Staubli VAL3: goHome.pjx

--- goHome.pjx ---
Parameters version=s7.8.3 stackSize=5000 millimeterUnit=true
Program file=_getP2PAngle.pgx
Program file=_getP2PDistance.pgx
Program file=_IsUseingBox.pgx
Program file=compteBox1Value.pgx
Program file=delete.pgx
Program file=editBigData.pgx
Program file=editSmlData.pgx
Program file=FCheckInBox1Pos.pgx
Program file=FCheckInBox2Pos.pgx
Program file=find.pgx
Program file=findInWhichBox1.pgx
Program file=FNearJt.pgx
Program file=getBoxSize.pgx
Program file=getEvent.pgx
Program file=getListTitle.pgx
Program file=getSizeItem.pgx
Program file=getTrajTool.pgx
Program file=GOHOME.pgx
Program file=goTo.pgx
Program file=HMI_setNewValue.pgx
Program file=HMI_setValue.pgx
Program file=initToSafePt.pgx
Program file=IsInTheSameBox.pgx
Program file=IsSetValue.pgx
Program file=IsUseSameTool.pgx
Program file=J_goTo.pgx
Program file=J_MoveTo.pgx
Program file=listAdd.pgx
Program file=loadMarkData.pgx
Program file=mark_All_Item.pgx
Program file=markItem.pgx
Program file=MoveTo.pgx
Program file=new.pgx
Program file=onSave.pgx
Program file=reveMarkItem.pgx
Data file=goHome.dtx
Library alias=sml path=./saveHomeBox/type1/type1.pjx
Library alias=big path=./saveHomeBox/type2/type2.pjx
Library alias=save path=./saveHomeBox/saveHomeBox.pjx
Library alias=language2 path=./language/language.pjx
Library alias=trajPt path=Disk://session/default/saveTraj/TRAJ/TRAJ.pjx
Library alias=saveData path=Disk://saveData/saveData.pjx
Library alias=jPt path=Disk://session/default/saveTraj/JPOINT/JPOINT.pjx
Library alias=use path=./userPage/userPage.pjx
Library alias=cycleStatus path=Disk://cycleStatus/cycleStatus.pjx
Library alias=tcp path=Disk://kernel/tool/tool.pjx
Library alias=language path=Disk://kernel/language/language.pjx
Library alias=jHome path=Disk://session/default/saveTraj/HOME/HOME.pjx
Type name=TrajSmallBox path=./template/TrajSmallBox/TrajSmallBox.pjx
Type name=TrajBigBox path=./template/TrajBigBox/TrajBigBox.pjx
Type name=TrajJoint path=Disk://kernel/template/TrajJoint/TrajJoint.pjx
Type name=Traies path=Disk://kernel/template/Traies/Traies.pjx

--- goHome.dtx ---
public TrajBigBox pRunBigPt
  [0]
    bool bJtEnabCheck[6]
    bool bMoveJHomeJoint
    bool bPosEnabCheck[3]
    jointRx jToHome
    num nIndexGun
    num nRobCtrlAreaNum[6]
    num nRobCtrlHJtsNum[12]
public TrajJoint tTrajJoint
  [0]
    num nIndexFrame
    num nIndexTool
    string sID = "qwer"
    TrajJointItem tData[2]
      [0]
        jointRx jJoint = {j1=-15.581719, j2=14.249611, j3=85.047741, j5=80.702759, j6=3.379944}
        TrajectoryItem tSuper
          [0]
            string comment
            num distance
            InstrItem iInstr[3]
              [0]
                string sData
                string sType
              [1]
                string sData
                string sType
              [2]
                string sData
                string sType
            num moveType
            num nMoveId
            num nStop
            num nTcpAction
            num nTime
            mdesc nom_speed = {tmax=9999, rmax=9999, leave=30, reach=30}
            bool toStop
      [1]
        jointRx jJoint = {j1=21.410587, j2=14.249611, j3=85.047741, j5=80.702759, j6=3.379944}
        TrajectoryItem tSuper
          [0]
            string comment
            num distance
            InstrItem iInstr[3]
              [0]
                string sData
                string sType
              [1]
                string sData
                string sType
              [2]
                string sData
                string sType
            num moveType
            num nMoveId
            num nStop
            num nTcpAction
            num nTime
            mdesc nom_speed = {tmax=9999, rmax=9999, leave=30, reach=30}
            bool toStop
public TrajSmallBox pRunSmlPt
  [0]
    bool bMountOnWall
    bool bMoveJHomeJoint
    bool bReverse_Tool_Z
    string comment
    jointRx jToHome
    num nIndexGun
    num nKeySafeNum[6]
    num nRe_Tool_Z_Dits
    num nRe_Tool_Z_WrdX
    num nRe_Tool_Z_WrdY
    num nRe_Tool_Z_WrdZ
    num nToSafeFrmX
    num nToSafeFrmY
    num nToSafeFrmZ
    num nToSafePtType
    num nTolKeySafeNum[6]
    pointRx pPointRx
    pointRx pToSafePt
    num nToolType
public bool bWizard
public pointRx pPointRx = {x=539.985307, y=-152.401921, z=239.262224, rx=-0.000498, ry=179.999963, rz=-12.063425, fatherId=world[0]}
tool tTool = {fatherId=flange[0], ioLink=valve1}
num nSelected
string sEvent
string sList
bool bRefresh
bool bSelected
num nKey
num nIndex
num nView
string sMessage
public string sMenu[8]
num nRefresh
num nTime = 1
string sTitle
num nOldIndex
num nOldLine
bool bFaceA
public string sJointLimt[6]
public string sFrmRob[6]
bool bLocked
bool bFindInBox1
public string sHomingStatus
public string sBox1
public string sBox2
public mdesc mHomeSpd = {accel=10, vel=10, decel=10, blend=off}
num nSign
num nCurrentUseType
num nInWhichBox
num nShortP2PDists
num nShortP2PAngle
bool bSetMax
public Traies tTraies
  [0]
    frame fFrame
    num nIndexTool
    string sID
    num nIndexFrame
    TrajItem tData
      [0]
        TrajectoryItem tSuper
          [0]
            num distance
            num moveType
            num nTime
            num nStop
            num nTcpAction
            string comment
            bool toStop
            mdesc nom_speed = {vel=450, tmax=1000}
            InstrItem iInstr[3]
              [0]
                string sType
                string sData
              [1]
                string sType
                string sData
              [2]
                string sType
                string sData
            num nMoveId
        pointRx pPoint
        num nType
        pointRx pCircle

--- _getP2PAngle.pgx ---
public program _getP2PAngle(point x_pHere, point x_pPoint, num& x_nP2PMaxAng[])
  local num l_nResult[14]
begin
  l_nResult[0]=abs(x_pPoint.trsf.rx-x_pHere.trsf.rx)
  l_nResult[1]=abs(x_pPoint.trsf.ry-x_pHere.trsf.ry)
  l_nResult[2]=min(l_nResult[0],360-l_nResult[0])
  l_nResult[3]=min(l_nResult[1],360-l_nResult[1])
  x_nP2PMaxAng=(l_nResult[2]+l_nResult[3])
end

--- _getP2PDistance.pgx ---
public program _getP2PDistance(point x_pPoint, point x_pHere, num& x_nP2PDsts[])
  local num l_nResult[14]
begin
  x_nP2PDsts=distance(position(x_pPoint,world),position(x_pHere,world))

end

--- _IsUseingBox.pgx ---
public program _IsUseingBox(bool& x_bNothing[])
  local string l_sEmpty
begin
  x_bNothing=true

  if  first(sml:box)!="" or first(big:box)!=""
    x_bNothing=false
  endIf
end

--- compteBox1Value.pgx ---
public program compteBox1Value(string x_sName, num& x_nKeySafeNum[])
  local num i
begin
  x_nKeySafeNum[0]=9999
  x_nKeySafeNum[1]=9999
  x_nKeySafeNum[2]=9999
  x_nKeySafeNum[3]=-9999
  x_nKeySafeNum[4]=-9999
  x_nKeySafeNum[5]=-9999
  //得到最小X
  for i=0 to size(sml:box[x_sName].pPointRx)-1
    if sml:box[x_sName].pPointRx[i].trsf.x<x_nKeySafeNum[0] and left(sml:box[x_sName].comment[i],1)=="#"
      x_nKeySafeNum[0]=sml:box[x_sName].pPointRx[i].trsf.x
    endIf
  endFor
  //得到最小Y
  for i=0 to size(sml:box[x_sName].pPointRx)-1
    if sml:box[x_sName].pPointRx[i].trsf.y<x_nKeySafeNum[1] and left(sml:box[x_sName].comment[i],1)=="#"
      x_nKeySafeNum[1]=sml:box[x_sName].pPointRx[i].trsf.y
    endIf
  endFor
  //得到最小Z
  for i=0 to size(sml:box[x_sName].pPointRx)-1
    if sml:box[x_sName].pPointRx[i].trsf.z<x_nKeySafeNum[2] and left(sml:box[x_sName].comment[i],1)=="#"
      x_nKeySafeNum[2]=sml:box[x_sName].pPointRx[i].trsf.z
    endIf
  endFor
  //得到最大X
  for i=0 to size(sml:box[x_sName].pPointRx)-1
    if sml:box[x_sName].pPointRx[i].trsf.x>x_nKeySafeNum[3] and left(sml:box[x_sName].comment[i],1)=="#"
      x_nKeySafeNum[3]=sml:box[x_sName].pPointRx[i].trsf.x
    endIf
  endFor
  //得到最大Y
  for i=0 to size(sml:box[x_sName].pPointRx)-1
    if sml:box[x_sName].pPointRx[i].trsf.y>x_nKeySafeNum[4] and left(sml:box[x_sName].comment[i],1)=="#"
      x_nKeySafeNum[4]=sml:box[x_sName].pPointRx[i].trsf.y
    endIf
  endFor
  //得到最大Z
  for i=0 to size(sml:box[x_sName].pPointRx)-1
    if sml:box[x_sName].pPointRx[i].trsf.z>x_nKeySafeNum[5] and left(sml:box[x_sName].comment[i],1)=="#"
      x_nKeySafeNum[5]=sml:box[x_sName].pPointRx[i].trsf.z
    endIf
  endFor
end

--- delete.pgx ---
public program delete(string x_sName (dimensions=1), num& x_nResult[] (dimensions=1))
  local num l_nSize
  local string l_sItem
begin
  //
  // delete the select option
  //
  if save:nBoxType==1
    if isDefined(sml:box[x_sName])
      // delete
      delete(sml:box[x_sName])
      // save it
      // bToSave=true
      x_nResult=0
    else
      x_nResult=-1
    endIf
  elseIf save:nBoxType==2
    if isDefined(big:box[x_sName])
      // delete
      delete(big:box[x_sName])
      // save it
      // bToSave=true
      x_nResult=0
    else
      x_nResult=-1
    endIf
  endIf
end

--- editBigData.pgx ---
public program editBigData(string x_sName, num& x_nResult)
  local string l_sMessage
  local string l_sEmpty
  local num i
  local string l_sItem
  local string l_sIsEanble[6]
  local num l_n
  local bool l_bOk
  local num l_nItemLow[6]
  local num l_nItemHigh[6]
  local num j
  local num l_nValue
  local string l_sFindEvent
  local num l_nValueMin
  local num l_nValueMax
  local string l_sEmpty1
  local num l_nMinX
  local num l_nMark
  local num l_nStep
  local bool l_bUnreached
  local num l_nMoveType
  local num l_nSize
  local string l_sInstruction
  local string l_sEvent
  local bool l_bFound
  local num l_nCount
  local bool l_bResult
  local string l_sButton[2]
  local joint l_jPoint
  local bool l_bPoint
  local tool l_tTool
begin
  nIndex=0
  use:nView=0
  cls()
  x_nResult=-1
  l_nStep=0
  //////////////////////////////////////
  bFaceA=true
  bSetMax=false
  if bWizard==true
     big:box[x_sName].jToHome[size(big:box[x_sName].jToHome)-1]=jHome:tTraj["home"].tData.jJoint[size(jHome:tTraj["home"].tData)-1]
     big:box[x_sName].nIndexGun=saveData:nIndexTool
  endIf
  while l_nStep<10
    switch l_nStep
      case -1
        x_nResult=-1
        resetMotion()
        return
      break
      case 0
        call language2:message(sMessage,69)
        title(sMessage)
        do
          if bFaceA
            cls()
            call use:type(31,13,"<<")
            call use:type(36,13,">>")
            call use:setSizeList(21,1,17,6)
            call use:setView(false)
            call language2:message(l_sItem,62)
            call use:listcreate(l_sItem)
            for l_n=0 to 5
              if big:box[x_sName].bPosEnabCheck[l_n]
                l_sIsEanble[l_n]=""
              else
                l_sIsEanble[l_n]="!"
              endIf
              l_nItemLow[l_n]=big:box[x_sName].nRobCtrlAreaNum[l_n*2]
              l_nItemHigh[l_n]=big:box[x_sName].nRobCtrlAreaNum[l_n*2+1]
            endFor

            sFrmRob[0]="<Rob_X<"
            sFrmRob[1]="<Rob_Y<"
            sFrmRob[2]="<Rob_Z<"
            sFrmRob[3]="<Rob_RX<"
            sFrmRob[4]="<Rob_RY<"
            sFrmRob[5]="<Rob_RZ<"
            for l_n=0 to 5
              sFrmRob[l_n]=l_sIsEanble[l_n]+toString("",l_nItemLow[l_n])+sFrmRob[l_n]+toString("",l_nItemHigh[l_n])
            endFor
            call use:listadd(sFrmRob)
            call use:listupdate1(0)
            //////////////////////////////////////
            call use:setSizeList(0,1,17,6)
            call use:setView(false)
            call language2:message(l_sItem,63)
            call use:listcreate(l_sItem)
            for l_n=0 to 5
              if big:box[x_sName].bJtEnabCheck[l_n]
                l_sIsEanble[l_n]=""
              else
                l_sIsEanble[l_n]="!"
              endIf
              l_nItemLow[l_n]=big:box[x_sName].nRobCtrlHJtsNum[l_n*2]
              l_nItemHigh[l_n]=big:box[x_sName].nRobCtrlHJtsNum[l_n*2+1]
            endFor
            sJointLimt[0]="<joint1<"
            sJointLimt[1]="<joint2<"
            sJointLimt[2]="<joint3<"
            sJointLimt[3]="<joint4<"
            sJointLimt[4]="<joint5<"
            sJointLimt[5]="<joint6<"
            for l_n=0 to 5
              sJointLimt[l_n]=l_sIsEanble[l_n]+toString("",l_nItemLow[l_n])+sJointLimt[l_n]+toString("",l_nItemHigh[l_n])
            endFor
            call use:listadd(sJointLimt)
            call use:listupdate(0)
            if !bSetMax
              i=get()
            endIf
            call use:listevent(i,nIndex,sEvent)
            if i==268
              bFaceA=false
            endIf
            delay(0)
          else
            cls()
            call use:type(30,13,"<<")
            call use:type(35,13,">>")
            call use:setSizeList(0,1,17,6)
            call use:setView(false)
            call language2:message(l_sItem,63)
            call use:listcreate(l_sItem)
            for l_n=0 to 5
              if big:box[x_sName].bJtEnabCheck[l_n]
                l_sIsEanble[l_n]=""
              else
                l_sIsEanble[l_n]="!"
              endIf
              l_nItemLow[l_n]=big:box[x_sName].nRobCtrlHJtsNum[l_n*2]
              l_nItemHigh[l_n]=big:box[x_sName].nRobCtrlHJtsNum[l_n*2+1]
            endFor
            sJointLimt[0]="<joint1<"
            sJointLimt[1]="<joint2<"
            sJointLimt[2]="<joint3<"
            sJointLimt[3]="<joint4<"
            sJointLimt[4]="<joint5<"
            sJointLimt[5]="<joint6<"
            for l_n=0 to 5
              sJointLimt[l_n]=l_sIsEanble[l_n]+toString("",l_nItemLow[l_n])+sJointLimt[l_n]+toString("",l_nItemHigh[l_n])
            endFor
            call use:listadd(sJointLimt)
            call use:listupdate1(0)
            /////////////////////////////////
            call use:setSizeList(21,1,17,6)
            call use:setView(false)
            call language2:message(l_sItem,62)
            call use:listcreate(l_sItem)
            for l_n=0 to 5
              if big:box[x_sName].bPosEnabCheck[l_n]
                l_sIsEanble[l_n]=""
              else
                l_sIsEanble[l_n]="!"
              endIf
              l_nItemLow[l_n]=big:box[x_sName].nRobCtrlAreaNum[l_n*2]
              l_nItemHigh[l_n]=big:box[x_sName].nRobCtrlAreaNum[l_n*2+1]
            endFor
            sFrmRob[0]="<Rob_X<"
            sFrmRob[1]="<Rob_Y<"
            sFrmRob[2]="<Rob_Z<"
            sFrmRob[3]="<Rob_RX<"
            sFrmRob[4]="<Rob_RY<"
            sFrmRob[5]="<Rob_RZ<"
            for l_n=0 to 5
              sFrmRob[l_n]=l_sIsEanble[l_n]+toString("",l_nItemLow[l_n])+sFrmRob[l_n]+toString("",l_nItemHigh[l_n])
            endFor
            call use:listadd(sFrmRob)
            call use:listupdate(0)
            if !bSetMax
              i=get()
            endIf
            call use:listevent(i,nIndex,sEvent)
            if i==264
              bFaceA=true
            endIf
            delay(0)
          endIf
          if i==278
            l_nStep=l_nStep+1
            l_bOk=true
          endIf
          if i==277
            x_nResult=-1
            wait(getKey()==-1)
            resetMotion( )
            return
          endIf
          if i==32
            if !bFaceA
              big:box[x_sName].bPosEnabCheck[nIndex]=!big:box[x_sName].bPosEnabCheck[nIndex]
            else
              big:box[x_sName].bJtEnabCheck[nIndex]=!big:box[x_sName].bJtEnabCheck[nIndex]
            endIf
          endIf
          if i==270 or bSetMax==true
            call use:listcursor(use:nView,false)
            if bFaceA==true
              if bSetMax==false
                l_nValueMin=big:box[x_sName].nRobCtrlHJtsNum[nIndex*2]

                if big:box[x_sName].bJtEnabCheck[nIndex]==true
                  l_nMinX=1
                else
                  l_nMinX=1+1
                endIf
                call HMI_setValue(l_nValueMin,0,0,l_nMinX,2+nIndex,l_sEmpty1)
                big:box[x_sName].nRobCtrlHJtsNum[nIndex*2]=l_nValueMin
                bSetMax=true
              else
                /////////////////////////////////////////////////////////////
                l_nValueMax=big:box[x_sName].nRobCtrlHJtsNum[nIndex*2+1]
                l_sFindEvent="joint"+toString("",nIndex+1)+"<"
                call use:findPos(sEvent,l_sFindEvent,j)
                call HMI_setValue(l_nValueMax,0,0,j+8,2+nIndex,l_sEmpty1)
                big:box[x_sName].nRobCtrlHJtsNum[nIndex*2+1]=l_nValueMax
                bSetMax=false
              endIf
            else
              if bSetMax==false
                l_nValueMin=big:box[x_sName].nRobCtrlAreaNum[nIndex*2]

                if big:box[x_sName].bPosEnabCheck[nIndex]==true
                  l_nMinX=22
                else
                  l_nMinX=22+1
                endIf
                call HMI_setValue(l_nValueMin,0,0,l_nMinX,2+nIndex,l_sEmpty1)
                big:box[x_sName].nRobCtrlAreaNum[nIndex*2]=l_nValueMin
                bSetMax=true
              else
                /////////////////////////////////////////////////////////////
                l_nValueMax=big:box[x_sName].nRobCtrlAreaNum[nIndex*2+1]
                l_sFindEvent="Rob"
                call use:findPos(sEvent,l_sFindEvent,j)
                if nIndex<=2
                  l_nMark=6
                else
                  l_nMark=7
                endIf
                call HMI_setValue(l_nValueMax,0,0,j+l_nMark+22,2+nIndex,l_sEmpty1)
                big:box[x_sName].nRobCtrlAreaNum[nIndex*2+1]=l_nValueMax
                bSetMax=false
              endIf
            endIf
          endIf
          i=-1
        until l_bOk==true
      break
       case 1
        if !cycleStatus:bCycle
          resetMotion( )
        endIf
        cls()
        call use:nullKey(nKey)
        call language2:message(sMessage,70)
        title(sMessage)
        //******************************************//
        bRefresh=true
        bSelected=false
        nIndex=0
        do
          do
            if big:box[x_sName].bMoveJHomeJoint[nIndex]
              l_nMoveType=1
            else
              l_nMoveType=0
            endIf
            call getTrajTool(l_tTool,big:box[x_sName].nIndexGun)
            call J_goTo(big:box[x_sName].jToHome[nIndex],nIndex,l_bUnreached,x_sName,l_nMoveType,l_tTool)
            if l_bUnreached
              // show the message out of range
              call language2:message(sMessage,51)
              call use:timerDialog(sMessage,1)
              l_bUnreached=false
              cls()
              bRefresh=true
            endIf
            if bRefresh==true
              bRefresh=false
              //******************bulid list*****************//
              l_sEmpty=""
              call use:stringCopy(l_sEmpty,sList)
              // Build the list
              l_nSize=size(big:box[x_sName].jToHome)
              for i=0 to l_nSize-1
                if big:box[x_sName].bMoveJHomeJoint[i]
                  call language2:message(l_sItem,46)
                else
                  call language2:message(l_sItem,45)
                endIf
                call language2:message(sMessage,44)
                l_sInstruction=toString("2",i+1)+" "+sMessage+" "+l_sItem
                call listAdd(l_sInstruction)
                l_sEvent=sList[i]
                if l_sEvent!=""
                  l_bFound=true
                  // update the selected item
                  if l_sEvent==sEvent
                    // nSelected=l_nCount
                  endIf
                  // add
                  if l_bFound
                    l_nCount=l_nCount+1
                  endIf
                endIf
              endFor
              cls()
              // define your list size for default
              call use:setSizeList(16,0,22,11)
              call use:setView(false)
              call language2:message(sMessage,43)
              call use:listcreate(sMessage)
              call use:listadd(sList)
              call language2:page(sMessage,304)
              call use:stringToArray(sMessage,sMenu)
              call use:setMenu(sMenu,true,3)
              // refresh the list
              call use:selectNewField(nSelected,nIndex,nView)

            else

            endIf
            nKey=getKey()
            call use:listevent(nKey,nIndex,sEvent)
            nView=use:nView
            nSelected=nIndex
            switch nKey
              case 271
                call language:getYesNo(l_sButton)
                call language2:message(sMessage,47)
                call use:yes_no(sMessage+"?",l_sButton,l_bResult)
                if l_bResult==true
                  big:box[x_sName].jToHome[nIndex]=herej()
                endIf
                bRefresh=true
                call use:nullKey(nKey)
              break
              case 272
                l_jPoint=big:box[x_sName].jToHome[nIndex]
                l_bPoint=big:box[x_sName].bMoveJHomeJoint[nIndex]
                insert(big:box[x_sName].jToHome[nIndex+1])
                insert(big:box[x_sName].bMoveJHomeJoint[nIndex+1])
                big:box[x_sName].jToHome[nIndex+1]=l_jPoint
                big:box[x_sName].bMoveJHomeJoint[nIndex+1]=l_bPoint
                bRefresh=true
                nSelected=nIndex+1
                call use:nullKey(nKey)
              break
              case 273
                if size(big:box[x_sName].jToHome)>1
                  call language:getYesNo(l_sButton)
                  call language2:message(sMessage,48)
                  call use:yes_no(sMessage+"?",l_sButton,l_bResult)
                  if l_bResult==true
                    delete(big:box[x_sName].jToHome[nIndex])
                    delete(big:box[x_sName].bMoveJHomeJoint[nIndex])
                    if nIndex>0
                      nIndex=nIndex-1
                      nSelected=nIndex-1
                    endIf
                  endIf
                  bRefresh=true
                endIf
                call use:nullKey(nKey)
              break
              case 274
                big:box[x_sName].bMoveJHomeJoint[nIndex]=!big:box[x_sName].bMoveJHomeJoint[nIndex]
                bRefresh=true
                call use:nullKey(nKey)
              break
              case 277
                l_nStep=l_nStep-1
                bRefresh=true
                bSelected=true
                call use:nullKey(nKey)
              break
              case 278
                bRefresh=true
                bSelected=true
                call use:nullKey(nKey)
                x_nResult=0
                if !cycleStatus:bCycle
                  resetMotion( )
                endIf
                return
              break
            endSwitch
            delay(0)
          until  bRefresh==true
        until  bSelected==true
        bSelected=false
    break
    endSwitch
  endWhile
  call use:nullKey(nKey)
  x_nResult=0
end

--- editSmlData.pgx ---
public program editSmlData(string x_sName, num& x_nResult)
  local num l_nStep
  local string l_sButton[2]
  local num i
  local string l_sEvent
  local bool l_bFound
  local num l_nCount
  local string l_sEmpty
  local num l_nSize
  local string l_sInstruction
  local bool l_bUnreached
  local num l_nResult
  local bool l_bResult
  local string l_sMessage[6]
  local bool l_bOk
  local bool l_bSelected
  local string l_sMountMsg
  local string l_sMessage1[3]
  local string l_sMessage2[2]
  local point l_pPoint
  local num l_nMoveType
  local joint l_jPoint
  local bool l_bPoint
  local string l_sItem
  local tool l_tTool
begin
  l_nStep=0
  call getTrajTool(tTool,sml:box[x_sName].nIndexGun)
  if bWizard==true
    call mark_All_Item(x_sName)
    call compteBox1Value(x_sName,sml:box[x_sName].nKeySafeNum)
    sml:box[x_sName].nToSafePtType=1
    sml:box[x_sName].nToolType=1
    call initToSafePt(x_sName)
    //初始推荐值
    if !sml:box[x_sName].bMountOnWall
      //地装推荐值为最大Z值
      sml:box[x_sName].nToSafeFrmZ=roundUp( sml:box[x_sName].nKeySafeNum[5])
      sml:box[x_sName].nRe_Tool_Z_WrdZ=roundUp( sml:box[x_sName].nKeySafeNum[5])
    else
      sml:box[x_sName].nToSafeFrmZ=roundUp( sml:box[x_sName].nKeySafeNum[2])
      sml:box[x_sName].nRe_Tool_Z_WrdZ=roundUp( sml:box[x_sName].nKeySafeNum[2])
    endIf
    sml:box[x_sName].jToHome[size(sml:box[x_sName].jToHome)-1]=jHome:tTraj["home"].tData.jJoint[size(jHome:tTraj["home"].tData)-1]
  endIf
  bSelected=false
  // WIZARD
  while l_nStep<10
    switch l_nStep
      case -1
        x_nResult=-1
        return
      break
      case 0
        if !cycleStatus:bCycle
          resetMotion( )
        endIf
        cls()
        l_bSelected=false
        l_bOk=false
        call language2:message(sMessage,27)
        title(sMessage)
        do
          do
            call language2:message(sMessage,11)
            l_sButton[0]=sMessage
            call use:type(0,13,sMessage)
            call language2:message(sMessage,12)
            l_sButton[1]=sMessage
            call use:type(5,13,sMessage)
            call use:type(30,13,"<<")
            call use:type(35,13,">>")
            call language2:message(sMessage,26)
            call use:type(1,1,sMessage+l_sButton[sel(sml:box[x_sName].bMountOnWall,1,0)])
            call language2:message(sMessage,10)
            call use:timerDialog(sMessage,0)
            nKey=get( )
            if nKey==278
              l_bOk=true
              l_nStep=l_nStep+1
              l_bSelected=true
            elseIf nKey==277
              x_nResult=-1
              call use:nullKey(nKey)
              return
            elseIf nKey==271
              l_bOk=true
              sml:box[x_sName].bMountOnWall=false
            elseIf nKey==272
              l_bOk=true
              sml:box[x_sName].bMountOnWall=true
            endIf
            delay(0)
          until l_bOk
        until l_bSelected
        call use:nullKey(nKey)
      break
      case 1
        //******************************************//
        call language2:message(sMessage,28)
        title(sMessage)
        bRefresh=true
        nIndex=0
        if !cycleStatus:bCycle
          resetMotion( )
        endIf
        do
          call goTo(sml:box[x_sName].pPointRx[nIndex],nIndex,l_bUnreached,x_sName,0)
          if l_bUnreached
            // show the message out of range
            call language2:message(sMessage,51)
            call use:timerDialog(sMessage,1)
            l_bUnreached=false
            cls()
            bRefresh=true
          endIf
          if bRefresh==true

            bRefresh=false
            //******************bulid list*****************//
            l_sEmpty=""
            call use:stringCopy(l_sEmpty,sList)
            // Build the list
            call getSizeItem(x_sName,l_nSize,0)
            for i=0 to l_nSize-1
              l_sInstruction=toString("2",i+1)+" "+sml:box[x_sName].comment[i]
              call listAdd(l_sInstruction)

            endFor
            cls()
            //set menu
            call language2:page(sMessage,302)
            call use:stringToArray(sMessage,sMenu)
            call use:setMenu(sMenu,true,3)
            // define your list size for default
            call use:setSizeList(16,0,22,11)
            call use:setView(false)
            call getListTitle(sTitle)
            call use:listcreate(x_sName)
            call use:listadd(sList)
            // refresh the list
            call use:selectNewField(nSelected,nIndex,nView)

          else

          endIf
          nKey=getKey()
          call use:listevent(nKey,nIndex,sEvent)
          nView=use:nView
          nSelected=nIndex
          switch nKey
            case 271
              if sEvent!=""
                call markItem(nIndex,x_sName)
                nSelected=nIndex+1
                bRefresh=true
              endIf
              call use:nullKey(nKey)
            break
            case 272
              if sEvent!=""
                call mark_All_Item(x_sName)
                bRefresh=true
              endIf
              call use:nullKey(nKey)
            break
            case 273
              if sEvent!=""
                call reveMarkItem(x_sName)
                bRefresh=true
              endIf
              call use:nullKey(nKey)
            break
            case 277
              l_nStep=0
              bSelected=true
              call use:nullKey(nKey)
            break
            case 278
              call language:getYesNo(l_sButton)
              call language2:message(sMessage,24)
              call use:yes_no(sMessage,l_sButton,l_bResult)
              if l_bResult==true
                l_nStep=2
                bSelected=true
              else
                bRefresh=true
              endIf
              call use:nullKey(nKey)
            break
          endSwitch

          delay(0)
        until  bSelected==true
        bSelected=false
      break
      case 2
        if !cycleStatus:bCycle
          resetMotion()
        endIf
        cls()
        call language2:message(sMessage,29)
        title(sMessage)
        call use:type(30,13,"<<")
        call use:type(35,13,">>")
        nIndex=0
        use:nView=0
        call compteBox1Value(x_sName,sml:box[x_sName].nKeySafeNum)
        do
          call use:setSizeList(20,2,18,6)
          call use:setView(false)
          call language2:message(sMessage,13)
          call use:listcreate(sMessage)
          call language2:message(sMessage,21)
          l_sMessage[0]=sMessage+"X:"+toString(".3",sml:box[x_sName].nKeySafeNum[0])+" mm"
          l_sMessage[1]=sMessage+"Y:"+toString(".3",sml:box[x_sName].nKeySafeNum[1])+" mm"
          l_sMessage[2]=sMessage+"Z:"+toString(".3",sml:box[x_sName].nKeySafeNum[2])+" mm"
          call language2:message(sMessage,20)
          l_sMessage[3]=sMessage+"X:"+toString(".3",sml:box[x_sName].nKeySafeNum[3])+" mm"
          l_sMessage[4]=sMessage+"Y:"+toString(".3",sml:box[x_sName].nKeySafeNum[4])+" mm"
          l_sMessage[5]=sMessage+"Z:"+toString(".3",sml:box[x_sName].nKeySafeNum[5])+" mm"
          call use:listadd(l_sMessage)
          call use:listupdate(0)
          i=get()
          call use:listevent(i,nIndex,l_sEmpty)
          use:nView=nIndex
          if nIndex!=nOldLine
            nOldLine=nIndex
          endIf
          delay(0)
        until i==278 or i==277
        switch i
          case 278
            l_nStep= l_nStep+1
            wait(getKey()==-1)
          break
          case 277
            l_nStep= l_nStep-1
            wait(getKey()==-1)
          break
        endSwitch
      break
      case 3
        if !cycleStatus:bCycle
          resetMotion()
        endIf
        cls()
        call language2:message(sMessage,30)
        title(sMessage)
        call use:type(30,13,"<<")
        call use:type(35,13,">>")
        nIndex=0
        use:nView=0
        do
          call use:setSizeList(20,2,18,6)
          call use:setView(false)
          call language2:message(sMessage,14)
          call use:listcreate(sMessage)
          call language2:message(sMessage,22)
          l_sMessage[0]=sMessage+"X:"+toString(".3",sml:box[x_sName].nTolKeySafeNum[0])+" mm"
          l_sMessage[1]=sMessage+"Y:"+toString(".3",sml:box[x_sName].nTolKeySafeNum[1])+" mm"
          l_sMessage[2]=sMessage+"Z:"+toString(".3",sml:box[x_sName].nTolKeySafeNum[2])+" mm"
          call language2:message(sMessage,23)
          l_sMessage[3]=sMessage+"X:"+toString(".3",sml:box[x_sName].nTolKeySafeNum[3])+" mm"
          l_sMessage[4]=sMessage+"Y:"+toString(".3",sml:box[x_sName].nTolKeySafeNum[4])+" mm"
          l_sMessage[5]=sMessage+"Z:"+toString(".3",sml:box[x_sName].nTolKeySafeNum[5])+" mm"
          call use:listadd(l_sMessage)
          call use:listupdate(0)
          i=get()
          call use:listevent(i,nIndex,l_sEmpty)
          use:nView=nIndex
          if nIndex!=nOldLine
            nOldLine=nIndex
          endIf
          if i==270
            call language2:message(sMessage,25)
            call HMI_setNewValue(sml:box[x_sName].nTolKeySafeNum[nIndex],0,0,0,13,sMessage)
            cls()
            use:bUseRefresh=true
            call use:type(30,13,"<<")
            call use:type(35,13,">>")
          endIf
          delay(0)
        until i==278 or i==277
        switch i
          case 278
            l_nStep= l_nStep+1
            wait(getKey()==-1)
          break
          case 277
            l_nStep= l_nStep-1
            wait(getKey()==-1)
          break
        endSwitch
      break
      case 4
        if !cycleStatus:bCycle
          resetMotion()
        endIf
        call language2:message(sMessage,31)
        title(sMessage)
        cls()
        call use:type(30,13,"<<")
        call use:type(35,13,">>")
        nIndex=0
        use:nView=0
        do
          call use:type(30,13,"<<")
          call use:type(35,13,">>")
          call use:setSizeList(5,2,33,3)
          call use:setView(false)
          call language2:message(sMessage,16)
          call use:listcreate(sMessage)
          if sml:box[x_sName].bMountOnWall==false
            call language2:message(sMessage,11)
          else
            call language2:message(sMessage,12)
          endIf
          l_sMountMsg=" "+sMessage
          call language2:message(sMessage,34)
          if sml:box[x_sName].nToSafePtType==1
            l_sMessage1[0]="@ "+sMessage+toString("",sml:box[x_sName].nToSafeFrmZ)+" mm"+l_sMountMsg
          else
            l_sMessage1[0]=sMessage+toString("",sml:box[x_sName].nToSafeFrmZ)+" mm"+l_sMountMsg
          endIf
          if sml:box[x_sName].nToSafePtType==2
            if !sml:box[x_sName].bReverse_Tool_Z==true
              call language2:message(sMessage,35)
              l_sMessage1[1]="@ "+sMessage+toString("",sml:box[x_sName].nRe_Tool_Z_Dits)+" mm"
            else
              call language2:message(sMessage,36)
              l_sMessage1[1]="@ "+sMessage+toString("",sml:box[x_sName].nRe_Tool_Z_WrdZ)+" mm"
            endIf
          else
            if !sml:box[x_sName].bReverse_Tool_Z
              call language2:message(sMessage,35)
              l_sMessage1[1]=sMessage+toString("",sml:box[x_sName].nRe_Tool_Z_Dits)+" mm"
            else
              call language2:message(sMessage,36)
              l_sMessage1[1]=sMessage+toString("",sml:box[x_sName].nRe_Tool_Z_WrdZ)+" mm"
            endIf
          endIf
          call language2:message(sMessage,19)
          if sml:box[x_sName].nToSafePtType==3
            l_sMessage1[2]="@ "+sMessage
          else
            l_sMessage1[2]=sMessage
          endIf
          call use:listadd(l_sMessage1)
          call use:listupdate(0)
          i=get()
          call use:listevent(i,nIndex,l_sEmpty)
          use:nView=nIndex
          if nIndex!=nOldLine
            nOldLine=nIndex
          endIf
          if i==270
            sml:box[x_sName].nToSafePtType=nIndex+1
            if sml:box[x_sName].nToSafePtType==1
              call language2:message(sMessage,25)
              call HMI_setNewValue(sml:box[x_sName].nToSafeFrmZ,0,0,0,13,sMessage)
            endIf
            if sml:box[x_sName].nToSafePtType==2
              do
                call use:setSizeList(3,2,26,2)
                call use:setView(false)
                call use:listcreate("")
                call language2:message(sMessage,35)
                l_sMessage2[0]=sMessage
                call language2:message(sMessage,36)
                l_sMessage2[1]=sMessage
                call use:listadd(l_sMessage2)
                call use:listupdate(0)
                nKey=get()
                call use:listevent(nKey,nIndex,l_sEvent)
                switch nKey
                  case 270
                    /////////////////////////////
                    if nIndex==0
                      sml:box[x_sName].bReverse_Tool_Z=false
                    else
                      sml:box[x_sName].bReverse_Tool_Z=true
                    endIf
                  break
                endSwitch
              until nKey==270
              if nIndex==0
                call language2:message(sMessage,25)
                call HMI_setNewValue(sml:box[x_sName].nRe_Tool_Z_Dits,0,0,0,13,sMessage)
              else
                call language2:message(sMessage,25)
                call HMI_setNewValue(sml:box[x_sName].nRe_Tool_Z_WrdZ,0,0,0,13,sMessage)
              endIf
            endIf
            cls()
          endIf
          delay(0)
        until i==278 or i==277
        switch i
          case 278
            if sml:box[x_sName].nToSafePtType==3
              l_nStep=l_nStep+1
            else
              l_nStep=l_nStep+2
            endIf
            wait(getKey()==-1)
          break
          case 277
            l_nStep=l_nStep-1
            wait(getKey()==-1)
          break
        endSwitch
      break
      case 5
        if !cycleStatus:bCycle
          resetMotion( )
        endIf
        cls()
        call language2:message(sMessage,31)
        title(sMessage+"-1")
        call language2:message(sMessage,37)
        call HMI_setNewValue(sml:box[x_sName].nToolType,1,2,0,13,sMessage)
        delay(0)
        call use:nullKey(nKey)
        call language2:message(sMessage,31)
        title(sMessage+"-2")
        //******************************************//
        bRefresh=true
        bSelected=false
        nIndex=0
        do
          do
            call goTo(sml:box[x_sName].pToSafePt[nIndex],nIndex,l_bUnreached,x_sName,0)
            if l_bUnreached
              // show the message out of range
              call language2:message(sMessage,51)
              call use:timerDialog(sMessage,1)
              l_bUnreached=false
              cls()
              bRefresh=true
            endIf
            if bRefresh==true

              bRefresh=false
              //******************bulid list*****************//
              l_sEmpty=""
              call use:stringCopy(l_sEmpty,sList)
              // Build the list
              call getSizeItem(x_sName,l_nSize,1)
              for i=0 to l_nSize-1
                call language2:message(sMessage,39)
                call language2:message(l_sItem,45)
                l_sInstruction=toString("2",i+1)+" "+sMessage+" "+l_sItem
                call listAdd(l_sInstruction)
                l_sEvent=sList[i]
                if l_sEvent!=""
                  l_bFound=true
                  // update the selected item
                  if l_sEvent==sEvent
                    // nSelected=l_nCount
                  endIf
                  // add
                  if l_bFound
                    l_nCount=l_nCount+1
                  endIf
                endIf
              endFor
              cls()
              // define your list size for default
              call use:setSizeList(16,0,22,11)
              call use:setView(false)
              call language2:message(sMessage,42)
              call use:listcreate(sMessage)
              call use:listadd(sList)
              call language2:page(sMessage,303)
              call use:stringToArray(sMessage,sMenu)
              call use:setMenu(sMenu,true,3)
              // refresh the list
              call use:selectNewField(nSelected,nIndex,nView)

            else

            endIf
            nKey=getKey()
            call use:listevent(nKey,nIndex,sEvent)
            nView=use:nView
            nSelected=nIndex
            switch nKey
              case 271
                call language:getYesNo(l_sButton)
                call language2:message(sMessage,40)
                call use:yes_no(sMessage+"?",l_sButton,l_bResult)
                if l_bResult==true
                  sml:box[x_sName].pToSafePt[nIndex]=here(tTool,world)
                endIf
                bRefresh=true
                call use:nullKey(nKey)
              break
              case 272
                if sEvent!=""
                  l_pPoint=sml:box[x_sName].pToSafePt[nIndex]
                  insert(sml:box[x_sName].pToSafePt[nIndex+1])
                  sml:box[x_sName].pToSafePt[nIndex+1]=l_pPoint
                  bRefresh=true
                  nSelected=nIndex+1
                endIf
                call use:nullKey(nKey)
              break
              case 273
                if size(sml:box[x_sName].pToSafePt)>1
                  call language:getYesNo(l_sButton)
                  call language2:message(sMessage,41)
                  call use:yes_no(sMessage+"?",l_sButton,l_bResult)
                  if l_bResult==true
                    delete(sml:box[x_sName].pToSafePt[nIndex])
                    if nIndex>0
                      nIndex=nIndex-1
                      nSelected=nIndex-1
                    endIf
                  endIf
                  bRefresh=true
                endIf
                call use:nullKey(nKey)
              break
              case 277
                l_nStep=l_nStep-1
                bRefresh=true
                bSelected=true
                call use:nullKey(nKey)
              break
              case 278
                l_nStep=l_nStep+1
                bRefresh=true
                bSelected=true
                call use:nullKey(nKey)
              break
            endSwitch
            delay(0)
          until  bRefresh==true
        until  bSelected==true
        bSelected=false
      break
      case 6
        if !cycleStatus:bCycle
          resetMotion( )
        endIf
        cls()
        call use:nullKey(nKey)
        call language2:message(sMessage,32)
        title(sMessage)
        //******************************************//
        bRefresh=true
        bSelected=false
        nIndex=0
        do
          do
            if sml:box[x_sName].bMoveJHomeJoint[nIndex]
              l_nMoveType=1
            else
              l_nMoveType=0
            endIf
            call getTrajTool(l_tTool,sml:box[x_sName].nIndexGun)
            call J_goTo(sml:box[x_sName].jToHome[nIndex],nIndex,l_bUnreached,x_sName,l_nMoveType,l_tTool)
            if l_bUnreached
              // show the message out of range
              call language2:message(sMessage,51)
              call use:timerDialog(sMessage,1)
              l_bUnreached=false
              cls()
              bRefresh=true
            endIf
            if bRefresh==true

              bRefresh=false
              //******************bulid list*****************//
              l_sEmpty=""
              call use:stringCopy(l_sEmpty,sList)
              // Build the list
              call getSizeItem(x_sName,l_nSize,2)
              for i=0 to l_nSize-1
                if sml:box[x_sName].bMoveJHomeJoint[i]
                  call language2:message(l_sItem,46)
                else
                  call language2:message(l_sItem,45)
                endIf
                call language2:message(sMessage,44)
                l_sInstruction=toString("2",i+1)+" "+sMessage+" "+l_sItem
                call listAdd(l_sInstruction)
                l_sEvent=sList[i]
                if l_sEvent!=""
                  l_bFound=true
                  // update the selected item
                  if l_sEvent==sEvent
                    // nSelected=l_nCount
                  endIf
                  // add
                  if l_bFound
                    l_nCount=l_nCount+1
                  endIf
                endIf
              endFor
              cls()
              // define your list size for default
              call use:setSizeList(16,0,22,11)
              call use:setView(false)
              call language2:message(sMessage,43)
              call use:listcreate(sMessage)
              call use:listadd(sList)
              call language2:page(sMessage,304)
              call use:stringToArray(sMessage,sMenu)
              call use:setMenu(sMenu,true,3)
              // refresh the list
              call use:selectNewField(nSelected,nIndex,nView)

            else

            endIf
            nKey=getKey()
            call use:listevent(nKey,nIndex,sEvent)
            nView=use:nView
            nSelected=nIndex
            switch nKey
              case 271
                call language:getYesNo(l_sButton)
                call language2:message(sMessage,47)
                call use:yes_no(sMessage+"?",l_sButton,l_bResult)
                if l_bResult==true
                  sml:box[x_sName].jToHome[nIndex]=herej()
                endIf
                bRefresh=true
                call use:nullKey(nKey)
              break
              case 272
                l_jPoint=sml:box[x_sName].jToHome[nIndex]
                l_bPoint=sml:box[x_sName].bMoveJHomeJoint[nIndex]
                insert(sml:box[x_sName].jToHome[nIndex+1])
                insert(sml:box[x_sName].bMoveJHomeJoint[nIndex+1])
                sml:box[x_sName].jToHome[nIndex+1]=l_jPoint
                sml:box[x_sName].bMoveJHomeJoint[nIndex+1]=l_bPoint
                bRefresh=true
                nSelected=nIndex+1
                call use:nullKey(nKey)
              break
              case 273
                if size(sml:box[x_sName].jToHome)>1
                  call language:getYesNo(l_sButton)
                  call language2:message(sMessage,48)
                  call use:yes_no(sMessage+"?",l_sButton,l_bResult)
                  if l_bResult==true
                    delete(sml:box[x_sName].jToHome[nIndex])
                    delete(sml:box[x_sName].bMoveJHomeJoint[nIndex])
                    if nIndex>0
                      nIndex=nIndex-1
                      nSelected=nIndex-1
                    endIf
                  endIf
                  bRefresh=true
                endIf
                call use:nullKey(nKey)
              break
              case 274
                sml:box[x_sName].bMoveJHomeJoint[nIndex]=!sml:box[x_sName].bMoveJHomeJoint[nIndex]
                bRefresh=true
                call use:nullKey(nKey)
              break
              case 277
                if sml:box[x_sName].nToSafePtType==3
                  l_nStep=l_nStep-1
                else
                  l_nStep=l_nStep-2
                endIf
                bRefresh=true
                bSelected=true
                call use:nullKey(nKey)
              break
              case 278

                bRefresh=true
                bSelected=true
                call use:nullKey(nKey)
                x_nResult=0
                if !cycleStatus:bCycle
                  resetMotion( )
                endIf
                return
              break
            endSwitch
            delay(0)
          until  bRefresh==true
        until  bSelected==true
        bSelected=false
      break
    endSwitch
    delay(0)
  endWhile
end

--- FCheckInBox1Pos.pgx ---
public program FCheckInBox1Pos(tool t_tool, frame fr_frame, bool& b_inArea[], num& x_nKeyNum[], num& nTolKeyNum[])
// Pruefen ob Roboter innerhalb eines definierten Bereichs
  local trsf tr_here
  local point p_here
  local trsf tr_NegPos
  local trsf tr_PosPos
  local trsf tr_BoxPos1
  local trsf tr_BoxPos2
begin
  //Header
  if false
    //判断机器人是否属于所设定的空间盒子中
    //Parameter:
    //  p_BoxPos1: Position 1 (包括开始位置跟结束位置)
    //  p_BoxPos2: Position 2 (包括开始位置跟结束位置)
    //  b_inArea: 返回参数  true  : 机器人在矩形中
    //                          false : 机器人属于非矩形中
    //
  endIf
  //判断变量返回
  b_inArea=true
  p_here=here(t_tool,fr_frame)
  tr_here=p_here.trsf
  if (tr_here.x>(x_nKeyNum[3]+nTolKeyNum[3])) or (tr_here.y>(x_nKeyNum[4]+nTolKeyNum[4])) or (tr_here.z>(x_nKeyNum[5]+nTolKeyNum[5]))
    b_inArea=false
  endIf
  if (tr_here.x<(x_nKeyNum[0]-nTolKeyNum[0])) or (tr_here.y<(x_nKeyNum[1]-nTolKeyNum[1])) or (tr_here.z<(x_nKeyNum[2]-nTolKeyNum[2]))
    b_inArea=false
  endIf
end

--- FCheckInBox2Pos.pgx ---
public program FCheckInBox2Pos(tool t_tool, frame fr_frame, bool& b_inArea[], bool& x_bJtEnabCheck[], bool& x_bPosEnabCheck[], num& x_nRobCtrlJts[], num& x_nRobCtrlArea[])
// Pruefen ob Roboter innerhalb eines definierten Bereichs
  local trsf tr_here
  local point p_here
  local trsf tr_NegPos
  local trsf tr_PosPos
  local trsf tr_BoxPos1
  local trsf tr_BoxPos2
  local jointRx j_here
  local num i
  local num l_nItem[6]
begin
  //Header
  if false
    //判断机器人是否属于所设定的空间盒子中
    //Parameter:
    //  p_BoxPos1: Position 1 (包括开始位置跟结束位置)
    //  p_BoxPos2: Position 2 (包括开始位置跟结束位置)
    //  b_inArea: 返回参数  true  : 机器人在矩形中
    //                          false : 机器人属于非矩形中
    //
  endIf
  //判断变量返回
  b_inArea=true
  p_here=here(t_tool,fr_frame)
  j_here=herej()
  ///////////////////////////////////////////////////
  tr_here=p_here.trsf
  l_nItem[0]=j_here.j1
  l_nItem[1]=j_here.j2
  l_nItem[2]=j_here.j3
  l_nItem[3]=j_here.j4
  l_nItem[4]=j_here.j5
  l_nItem[5]=j_here.j6
  for i=0 to 5
    if x_bJtEnabCheck[i]
      if l_nItem[i]>=x_nRobCtrlJts[i*2+1] or l_nItem[i]<=x_nRobCtrlJts[i*2]
        b_inArea=false
      endIf
    endIf
  endFor
  /////////////////////////////////////////
  l_nItem[0]=p_here.trsf.x
  l_nItem[1]=p_here.trsf.y
  l_nItem[2]=p_here.trsf.z
  l_nItem[3]=p_here.trsf.rx
  l_nItem[4]=p_here.trsf.ry
  l_nItem[5]=p_here.trsf.rz
  for i=0 to 5
    if x_bPosEnabCheck[i]
      if l_nItem[i]>=x_nRobCtrlArea[i*2+1] or l_nItem[i]<=x_nRobCtrlArea[i*2]
        b_inArea=false
      endIf
    endIf
  endFor
end

--- find.pgx ---
public program find(string& x_sItem[] (dimensions=1), bool& x_bFound[] (dimensions=1))
begin
  // check if the item has been foundf
  if save:nBoxType==1
    x_bFound=isDefined(sml:box[x_sItem])
  elseIf save:nBoxType==2
    x_bFound=isDefined(big:box[x_sItem])
  endIf
end

--- findInWhichBox1.pgx ---
program findInWhichBox1(string& x_sLodaBox1[])
  local num i
  local num l_nResult
  local point l_pHere
  local tool l_tTool
  local num j
  local num k
  local num l_nAngle
  local num l_nPointIndex
  local num m
  local num l_nShort
  local bool l_bCondition
  local num l_nSize
begin

  //分析比较最可能的安全盒子
  l_nSize=size(nInWhichBox)
  resize(nShortP2PAngle,1,l_nSize)
  resize(nShortP2PDists,1,l_nSize)
  for k=0 to size(nShortP2PDists)-1
    nShortP2PAngle[k]=9999
    nShortP2PDists[k]=9999
  endFor
  for i=0 to size(nInWhichBox)-1


      call getTrajTool(l_tTool,sml:box[sBox1[i]].nIndexGun )
      l_pHere=here(l_tTool,world)
      l_bCondition=false
      for j=0 to size(sml:box[sBox1[i]].comment)-1
        if left(sml:box[sBox1[i]].comment[j],1)=="#"
          call _getP2PAngle(l_pHere,sml:box[sBox1[i]].pPointRx[j],l_nAngle)
          if nShortP2PAngle[i]>l_nAngle and l_nAngle<=15
            nShortP2PAngle[i]=l_nAngle
            l_bCondition=true
            l_nPointIndex=j
          endIf
        endIf
      endFor
      if l_bCondition
        call _getP2PDistance(sml:box[sBox1[i]].pPointRx[l_nPointIndex],l_pHere,nShortP2PDists[i])
      endIf

  endFor
  l_nShort=99999
  for m=0 to size(nShortP2PDists)-1
    if nShortP2PDists[m]<l_nShort
      l_nShort=nShortP2PDists[m]
      x_sLodaBox1=sBox1[nInWhichBox[m]]
    endIf

  endFor
end

--- FNearJt.pgx ---
public program FNearJt(joint j_Position, num n_Tolerance, bool& m_inRange[])
begin
  //判断当前位置是否在某关节点附近
  m_inRange=(abs(herej()-j_Position)<{1,1,1,2,2,2})

end

--- getBoxSize.pgx ---
public program getBoxSize(num x_nType (dimensions=1), num& x_nSize (dimensions=1))
  local string l_sLibList
begin
  //得到所有回HOME设置数据文件库大小
  switch x_nType
    case 1
      //small box size
      x_nSize=size(sml:box)
    break
    case 2
      //big box size
      x_nSize=size(big:box)
    break
  endSwitch
end

--- getEvent.pgx ---
public program getEvent(string& x_sItem, num x_nIndex, num x_nBoxType)
  local num i
  local string l_sKey
begin

  switch x_nBoxType
    case 1
      // start from the first
      l_sKey=first(sml:box)
      // search it
      while l_sKey!=""
        x_sItem=l_sKey
        l_sKey=next(sml:box[l_sKey])
        if i==x_nIndex
          return
        else
          i=i+1
        endIf
      endWhile
    break
    case 2
      // start from the first
      l_sKey=first(big:box)
      // search it
      while l_sKey!=""
        x_sItem=l_sKey
        l_sKey=next(big:box[l_sKey])
        if i==x_nIndex
          return
        else
          i=i+1
        endIf
      endWhile
    break
  endSwitch
end

--- getListTitle.pgx ---
public program getListTitle(string& x_sMsg (dimensions=1))
begin
  if save:nBoxType==1
    call language2:message(x_sMsg,1)
  elseIf save:nBoxType==2
    call language2:message(x_sMsg,2)
  endIf
end

--- getSizeItem.pgx ---
public program getSizeItem(string x_sName, num& x_nSize, num x_nType)
begin
  switch  x_nType
    case 0
      x_nSize=size(sml:box[x_sName].pPointRx)
    break
    case 1
      x_nSize=size(sml:box[x_sName].pToSafePt)
    break
    case 2
      x_nSize=size(sml:box[x_sName].jToHome)
    break
  endSwitch
end

--- getTrajTool.pgx ---
public program getTrajTool(tool& x_tTool[], num x_nIndex)
begin
  // get the traj tool
  call tcp:getTool(x_tTool,x_nIndex)
end

--- GOHOME.pgx ---
public program GOHOME()
  local bool l_bInBoxOK
  local bool l_bFindInbox
  local bool l_bInBox1
  local num l_nSize
  local num i
  local tool l_tTool
  local bool l_bInPos
  local bool l_bIsHome
  local string l_sLoadBox
  local point l_pHere
  local point l_pPoint
  local bool l_bReturnOK
  local num l_nCount
  local point l_pCurrent
  local num m
  local num k
  local string l_sItem
  local string l_sItem1
begin
  call language2:message(sHomingStatus,57)
  l_bFindInbox=false
  l_bInBox1=false
  l_bInBoxOK=false
  bFindInBox1=false
  resetMotion()
  //类型1搜索...
  call getBoxSize(1,l_nSize)
  if l_nSize!=0

    resize(bFindInBox1,1,l_nSize)
    resize(sBox1,1,l_nSize)
    sBox1=""

      for i=0 to l_nSize-1
        call getEvent(sBox1[i],i,1)
      endFor
       if sBox1!=""
      for i=0 to l_nSize-1
        call getTrajTool(l_tTool,sml:box[sBox1[i]].nIndexGun )
        call FCheckInBox1Pos(l_tTool,world,l_bInPos,sml:box[sBox1[i]].nKeySafeNum,sml:box[sBox1[i]].nTolKeySafeNum)
        if l_bInPos
          bFindInBox1[i]=true
          l_bInBoxOK=true
        else
          bFindInBox1[i]=false
        endIf

      endFor
      call FNearJt(jHome:tTraj["home"].tData.jJoint[size(jHome:tTraj["home"].tData)-1],3,l_bIsHome)
      if l_bInBoxOK and !l_bIsHome
        call IsInTheSameBox(bFindInBox1,l_sLoadBox,l_bInBox1)
        if l_bInBox1
          call getTrajTool(l_tTool,sml:box[l_sLoadBox].nIndexGun )
          //在设定的区域?
          call language2:message(l_sItem,55)
          call language2:message(l_sItem1,56)
          sHomingStatus=l_sItem+l_sLoadBox+l_sItem1
          switch sml:box[l_sLoadBox].nToSafePtType
            case 1
              l_bFindInbox=true
              l_pHere=here(l_tTool,world)
              l_pPoint=l_pHere
              l_pPoint.trsf.z=sml:box[l_sLoadBox].nToSafeFrmZ
              movel(l_pPoint,l_tTool,mHomeSpd)
              waitEndMove()
            break
            case 2
              l_bFindInbox=true
              if !sml:box[l_sLoadBox].bReverse_Tool_Z
                l_pHere=here(l_tTool,world)
                l_pPoint=appro(l_pHere,{0,0,-sml:box[l_sLoadBox].nRe_Tool_Z_Dits,0,0,0})
                movel(l_pPoint,l_tTool,mHomeSpd)
                waitEndMove()
              else
                l_bReturnOK=false
                if sml:box[l_sLoadBox].bMountOnWall==false
                  nSign=1
                else
                  nSign=-1
                endIf
                do
                  l_pHere=here(l_tTool,world)
                  if l_pHere.trsf.z<=sml:box[l_sLoadBox].nRe_Tool_Z_WrdZ
                    movel(appro(l_pHere,{0,0,-1*nSign*100,0,0,0}),l_tTool,mHomeSpd)
                    l_nCount=l_nCount+1
                    do
                      l_pCurrent=here(l_tTool,world)
                    until l_pCurrent.trsf.z>=sml:box[l_sLoadBox].nRe_Tool_Z_WrdZ or isEmpty()
                    if l_pCurrent.trsf.z>=sml:box[l_sLoadBox].nRe_Tool_Z_WrdZ
                      l_bReturnOK=true
                    endIf
                  else
                    movel(appro(l_pHere,{0,0,nSign*100,0,0,0}),l_tTool,mHomeSpd)
                    l_nCount=l_nCount+1
                    do
                      l_pCurrent=here(l_tTool,world)
                    until l_pCurrent.trsf.z<=sml:box[l_sLoadBox].nRe_Tool_Z_WrdZ or isEmpty()
                    if l_pCurrent.trsf.z<=sml:box[l_sLoadBox].nRe_Tool_Z_WrdZ
                      l_bReturnOK=true
                    endIf
                  endIf
                until l_nCount==10 or l_bReturnOK==true
                stopMove()
                resetMotion()
              endIf
            break
            case 3
              //              if nCurrentUseType==Box1Pts:nToolType
              l_bFindInbox=true
              for m=0 to size(sml:box[l_sLoadBox].pToSafePt)-1
                movel(sml:box[l_sLoadBox].pToSafePt[m],l_tTool,mHomeSpd)
              endFor
              //              endIf
            break
          endSwitch
          // if sml:box[l_sLoadBox].nToSafePtType!=3 or (sml:box[l_sLoadBox].nToSafePtType==3 and cycleStatus:nCurrentUseTool==Box1Pts:nToolType)
          //      if sml:box[l_sLoadBox].nToSafePtType!=3
          for k=0 to size(sml:box[l_sLoadBox].jToHome)-1
            if sml:box[l_sLoadBox].bMoveJHomeJoint[k]
              movej(sml:box[l_sLoadBox].jToHome[k],l_tTool,mHomeSpd)
            else
              l_pPoint=jointToPoint(l_tTool,world,sml:box[l_sLoadBox].jToHome[k])
              movel(l_pPoint,l_tTool,mHomeSpd)
            endIf
          endFor
          //      endIf
          waitEndMove()
        endIf
      endIf
    endIf
  endIf
  //类型2搜索...
  if  l_bFindInbox==false
    call getBoxSize(2,l_nSize)
    if l_nSize!=0
      resize(sBox2,1,l_nSize)
      sBox2=""
      for i=0 to l_nSize-1
        call getEvent(sBox2[i],i,2)
      endFor
      if sBox2!=""
        for i=0 to l_nSize-1
          l_sLoadBox=sBox2[i]
          call getTrajTool(l_tTool,big:box[l_sLoadBox].nIndexGun )
          call FCheckInBox2Pos(l_tTool,world,l_bInPos,big:box[l_sLoadBox].bJtEnabCheck,big:box[l_sLoadBox].bPosEnabCheck,big:box[l_sLoadBox].nRobCtrlHJtsNum,big:box[l_sLoadBox].nRobCtrlAreaNum)
          call FNearJt(jHome:tTraj["home"].tData.jJoint[size(jHome:tTraj["home"].tData)-1],3,l_bIsHome)
          if l_bInPos and !l_bIsHome
            //在设定的区域?
            call language2:message(l_sItem,68)
            call language2:message(l_sItem1,56)
            sHomingStatus=l_sItem+l_sLoadBox+l_sItem1
            l_bFindInbox=true
            for k=0 to size(big:box[l_sLoadBox].jToHome)-1
              if big:box[l_sLoadBox].bMoveJHomeJoint[k]
                movej(big:box[l_sLoadBox].jToHome[k],l_tTool,mHomeSpd)
              else
                l_pPoint=jointToPoint(l_tTool,world,big:box[l_sLoadBox].jToHome[k])
                movel(l_pPoint,l_tTool,mHomeSpd)
              endIf
            endFor
            waitEndMove()
          endIf

        endFor
      endIf
    endIf
  endIf
  if !l_bFindInbox
    call language2:message(sHomingStatus,67)
    delay(1)
  endIf
  cycleStatus:bHoming=false

  resetMotion()
end

--- goTo.pgx ---
program goTo(point x_pPoint, num x_nIndex, bool& x_bUnreached[], string x_sName, num x_nMoveType)
  local bool l_bUnreached
  local num l_nIndexTool
  local tool l_tTool
  local num l_nMoveType
  local mdesc l_mDesc
begin
  // look for not cycle mode
  if !cycleStatus:bCycle
    if cycleStatus:nWorkingMode==1 and isPowered()
      // check for the index
      if nOldIndex!=x_nIndex or (cycleStatus:nWorkingStatus!=0 and cycleStatus:nWorkingStatus!=6)
        if !isEmpty()
          resetMotion()
        endIf
        if nOldIndex!=x_nIndex
          nOldIndex=x_nIndex
        endIf
      else
        if isEmpty() and cycleStatus:nWorkingStatus==0
          // get the data to move
          call getTrajTool(l_tTool,sml:box[x_sName].nIndexGun)
          // use a sTemp mdesc to set the blend off
          l_mDesc.blend=off
          l_mDesc.accel=l_mDesc.decel=10
          l_mDesc.vel=10
          // use the got to of the trajectory...
          call MoveTo(x_pPoint,l_tTool,l_mDesc,x_nMoveType,x_bUnreached)
        endIf
      endIf
    else
      if cycleStatus:nWorkingMode!=1
        resetMotion()
      endIf
    endIf
  endIf
end

--- HMI_setNewValue.pgx ---
public program HMI_setNewValue(num& x_nValue, num x_nMin, num x_nMax, num x_nX, num x_nY, string& x_sItem)
  local bool l_bOk
  local bool l_bQuit
  local string l_sMessage
begin
  call use:clear(0,13)
  do
    do
      call use:setSizeList(x_nX,x_nY-2,23,1)
      call use:listcreate("")
      call use:type(35,13,"OK")
      gotoxy(x_nX+1,x_nY-1)
      put(x_sItem)
      do
        nKey=get(x_nValue)
      until nKey==270 or nKey==278
      if x_nMin==0 and x_nMax==0
        l_bOk=true
      elseIf  x_nValue>=x_nMin and x_nValue<=x_nMax
          l_bOk=true
      else
        call language2:message(l_sMessage,38)
        popUpMsg(l_sMessage)
      endIf

    until l_bOk
    if nKey==278
      l_bQuit=true
    endIf
    call use:nullKey(nKey)
  until l_bQuit
end

--- HMI_setValue.pgx ---
public program HMI_setValue(num& x_nValue, num x_nMin, num x_nMax, num x_nX, num x_nY, string& x_sItem)
  local bool l_bOk
  local bool l_bQuit
  local string l_sMessage
begin

    do
      gotoxy(x_nX,x_nY)
      put(x_sItem)
      do
        nKey=get(x_nValue)
      until nKey==270
      if x_nMin==0 and x_nMax==0
        l_bOk=true
      elseIf  x_nValue>=x_nMin and x_nValue<=x_nMax
          l_bOk=true
      else
        call language2:message(l_sMessage,38)
        popUpMsg(l_sMessage)
      endIf

    until l_bOk

    call use:nullKey(nKey)

end

--- initToSafePt.pgx ---
program initToSafePt(string x_sName)
  local num i
  local num j
  local num l_n
begin
  l_n=-9999
  for i=0 to size(sml:box[x_sName].pPointRx)-1
    if sml:box[x_sName].pPointRx[i].trsf.z>l_n and left(sml:box[x_sName].comment[i],1)=="#"
      j=i
    endIf
  endFor
  sml:box[x_sName].pToSafePt=sml:box[x_sName].pPointRx[j]
end

--- IsInTheSameBox.pgx ---
program IsInTheSameBox(bool& x_bFindInBox1[], string& x_sLodaBox1[], bool& x_bInBox1[])
  local num i
  local num l_nNum
begin
  l_nNum=1
  resize(nInWhichBox,1,1)
  nInWhichBox=-1
  for i=0 to size(x_bFindInBox1)-1
    if x_bFindInBox1[i]==true
      x_bInBox1=true
      if nInWhichBox[size(nInWhichBox)-1]==-1
        nInWhichBox=i
      else
        $dins(nInWhichBox,size(nInWhichBox))
        nInWhichBox[size(nInWhichBox)-1]=i
      endIf
    endIf
  endFor
  if size(nInWhichBox)==1
    x_sLodaBox1=sBox1[nInWhichBox]
  else
    call findInWhichBox1(x_sLodaBox1)
  endIf

end

--- IsSetValue.pgx ---
public program IsSetValue()
begin
  //  x_bOk=true
  //  if save:nBoxType==1
  //
  //    if  sml:box[x_sName].nKeySafeNum[0]==0
  //
  //
  //    endIf
  //  elseIf save:nBoxType==2
  //
  //  endIf
end

--- IsUseSameTool.pgx ---
public program IsUseSameTool(string& x_sCheck[], bool& x_bResult)
  local num i
  local string l_sEvent
  local tool l_tTool
  local tool l_tOldTool
begin
  l_tOldTool.trsf.x=-123456
  x_bResult=true
  for i=0 to size(x_sCheck)-1
    if left(x_sCheck[i],4)=="TRAJ"
      l_sEvent=right(x_sCheck[i],len(x_sCheck[i])-5)
      if isDefined(trajPt:tTraj[l_sEvent])
        // use the type...
        tTraies=trajPt:tTraj[l_sEvent]
      endIf
      call getTrajTool(l_tTool,tTraies.nIndexTool)

    endIf
    if left(x_sCheck[i],6)=="JPOINT"
      l_sEvent=right(x_sCheck[i],len(x_sCheck[i])-7)
      if isDefined(jPt:tTraj[l_sEvent])
        // use the type...
        tTrajJoint=jPt:tTraj[l_sEvent]
      endIf
      call getTrajTool(l_tTool,tTrajJoint.nIndexTool)
    endIf
    if l_tOldTool.trsf.x==-123456
      l_tOldTool=l_tTool
    else
      if l_tOldTool!=l_tTool
        x_bResult=false
        return
      endIf
    endIf
  endFor
end

--- J_goTo.pgx ---
program J_goTo(jointRx x_jPoint, num x_nIndex, bool& x_bUnreached[], string x_sName, num x_nMoveType, tool x_tTool)
  local bool l_bUnreached
  local num l_nIndexTool
  local tool l_tTool
  local num l_nMoveType
  local mdesc l_mDesc
begin
  // look for not cycle mode
  if !cycleStatus:bCycle
    if cycleStatus:nWorkingMode==1 and isPowered()
      // check for the index
      if nOldIndex!=x_nIndex or (cycleStatus:nWorkingStatus!=0 and cycleStatus:nWorkingStatus!=6)
        if !isEmpty()
          resetMotion()
        endIf
        if nOldIndex!=x_nIndex
          nOldIndex=x_nIndex
        endIf
      else
        if isEmpty() and cycleStatus:nWorkingStatus==0
          // get the data to move
          // use a sTemp mdesc to set the blend off
          l_mDesc.blend=off
          l_mDesc.accel=l_mDesc.decel=10
          l_mDesc.vel=10
          // use the got to of the trajectory...
          call J_MoveTo(x_jPoint,x_tTool,l_mDesc,x_nMoveType,x_bUnreached)
        endIf
      endIf
    else
      if cycleStatus:nWorkingMode!=1
        resetMotion()
      endIf
    endIf
  endIf
end

--- J_MoveTo.pgx ---
program J_MoveTo(jointRx x_jPoint, tool x_tTool, mdesc x_mDesc, num x_nMoveType, bool& x_bReached)
  local bool l_bReached
  local joint l_jJoint
begin

    switch x_nMoveType
      case 0
        if pointToJoint(x_tTool,herej(),jointToPoint(x_tTool,world,x_jPoint),l_jJoint)
          movel(jointToPoint(x_tTool,world,x_jPoint),x_tTool,x_mDesc)
        else
          x_bReached=true
        endIf
      break
      case 1
        movej(x_jPoint,x_tTool,x_mDesc)
      break
    endSwitch

  end

--- listAdd.pgx ---
program listAdd(string x_sEvent)
begin
  // add in the queue
  if sList!=""
    insert(sList[size(sList)])
  endIf
  sList[size(sList)-1]=x_sEvent
end

--- loadMarkData.pgx ---
public program loadMarkData(string x_sName, string& x_sMarkList[])
  local num i
  local num j
  local num l_nIndex
  local num l_nSize
  local point l_pPoint
  local string l_sEvent
  local tool l_tTool
begin
  // x_sMarkList

  for i=0 to size(x_sMarkList)-1
    if left(x_sMarkList[i],4)=="TRAJ"
      l_sEvent=right(x_sMarkList[i],len(x_sMarkList[i])-5)
      if isDefined(trajPt:tTraj[l_sEvent])
        // use the type...
        tTraies=trajPt:tTraj[l_sEvent]
      endIf
      l_nSize=size(tTraies.tData)
      for j=0 to l_nSize-1
        if l_nIndex!=0
          insert(sml:box[x_sName].pPointRx[size(sml:box[x_sName].pPointRx)])
          insert(sml:box[x_sName].comment[size(sml:box[x_sName].comment)])
        endIf
        l_pPoint=trajPt:tTraj[l_sEvent].tData[j].pPoint
        pPointRx.trsf=position(l_pPoint,world)
        link(sml:box[x_sName].pPointRx[l_nIndex],world)
        sml:box[x_sName].pPointRx[l_nIndex].trsf=pPointRx.trsf
        sml:box[x_sName].pPointRx[l_nIndex].config=l_pPoint.config
        sml:box[x_sName].comment[l_nIndex]=trajPt:tTraj[l_sEvent].tData[j].tSuper.comment
        l_nIndex=l_nIndex+1
      endFor
      if  sml:box[x_sName].nIndexGun!=tTraies.nIndexTool
        sml:box[x_sName].nIndexGun=tTraies.nIndexTool
      endIf
    endIf
    if left(x_sMarkList[i],6)=="JPOINT"
      l_sEvent=right(x_sMarkList[i],len(x_sMarkList[i])-7)
      if isDefined(jPt:tTraj[l_sEvent])
        // use the type...
        tTrajJoint=jPt:tTraj[l_sEvent]
      endIf
      l_nSize=size(tTrajJoint.tData)
      for j=0 to l_nSize-1
        if l_nIndex!=0
          insert(sml:box[x_sName].pPointRx[size(sml:box[x_sName].pPointRx)])
          insert(sml:box[x_sName].comment[size(sml:box[x_sName].comment)])
        endIf
        l_pPoint=jointToPoint(tTool,world,jPt:tTraj[l_sEvent].tData[j].jJoint)
        link(sml:box[x_sName].pPointRx[l_nIndex],world)
        sml:box[x_sName].pPointRx[l_nIndex].trsf=l_pPoint.trsf
        sml:box[x_sName].pPointRx[l_nIndex].config=l_pPoint.config
        sml:box[x_sName].comment[l_nIndex]=jPt:tTraj[l_sEvent].tData[j].tSuper.comment
        l_nIndex=l_nIndex+1
      endFor
      if  sml:box[x_sName].nIndexGun!=tTrajJoint.nIndexTool
        sml:box[x_sName].nIndexGun=tTrajJoint.nIndexTool
      endIf
    endIf
  endFor

end

--- mark_All_Item.pgx ---
program mark_All_Item(string x_sName)
  local num i
begin
  for i=0 to size(sml:box[x_sName].comment)-1
    if left(sml:box[x_sName].comment[i],1)!="#"
    sml:box[x_sName].comment[i]="# "+sml:box[x_sName].comment[i]
    endIf
  endFor
end

--- markItem.pgx ---
public program markItem(num x_nIndex, string x_sName)
begin
  if left(sml:box[x_sName].comment[x_nIndex],1)!="#"
    sml:box[x_sName].comment[x_nIndex]="# "+sml:box[x_sName].comment[x_nIndex]
  else
    sml:box[x_sName].comment[x_nIndex]=right(sml:box[x_sName].comment[x_nIndex],len(sml:box[x_sName].comment[x_nIndex])-2)
  endIf
end

--- MoveTo.pgx ---
program MoveTo(pointRx x_pPoint, tool x_tTool, mdesc x_mDesc, num x_nMoveType, bool& x_bUnReachable)
  local string l_sMessage
  local joint l_jJoint
begin
  if pointToJoint(x_tTool,herej(),x_pPoint,l_jJoint)
    switch x_nMoveType
      case 0
        movel(x_pPoint,x_tTool,x_mDesc)
      break
      case 1
        movej(x_pPoint,x_tTool,x_mDesc)
      break
    endSwitch
  else
     x_bUnReachable=true
  endIf
end

--- new.pgx ---
public program new(string x_sName (dimensions=1), num& x_nResult[] (dimensions=1))
  local num l_nResult
  local string l_sPrefix
begin
  // new one
  if save:nBoxType==1
    if insert(sml:box[x_sName])
      x_nResult=0
    else
      x_nResult=-1
    endIf
  elseIf save:nBoxType==2
    if insert(big:box[x_sName])
      x_nResult=0
    else
      x_nResult=-1
    endIf
  endIf
end

--- onSave.pgx ---
public program onSave()
begin
  sml:libSave()
  big:libSave()
end

--- reveMarkItem.pgx ---
public program reveMarkItem(string x_sName)
  local num i
begin
  for i=0 to size(sml:box[x_sName].comment)-1
    if left(sml:box[x_sName].comment[i],1)!="#"
      sml:box[x_sName].comment[i]="# "+sml:box[x_sName].comment[i]
    else
     sml:box[x_sName].comment[i]=right(sml:box[x_sName].comment[i],len(sml:box[x_sName].comment[i])-2)
    endIf
  endFor
end
